// TIA Portal V16 export
// export: Created 2022-11-17T11:55:28.2915288Z, ExportSetting WithDefaults, DisplayName Totally Integrated Automation Portal, DisplayVersion V16 Update 6, DisplayName TIA Portal Version Control Interface, DisplayVersion V16 Update 2, DisplayName TIA Portal Openness, DisplayVersion V16 Update 6, DisplayName SINAMICS Startdrive Advanced, DisplayVersion V16 Update 5, DisplayName SINAMICS Startdrive G130, G150, S120, S150, SINAMICS MV, S210, DisplayVersion V16 Update 5, DisplayName SINAMICS Startdrive G110M, G120, G120C, G120D, G120P, G115D, DisplayVersion V16 Update 5, DisplayName STEP 7 Professional, DisplayVersion V16 Update 6, DisplayName STEP 7 Safety, DisplayVersion V16, DisplayName WinCC Advanced, DisplayVersion V16 Update 6
DATA_BLOCK "DB22_DisplayData"   // DB22
{ S7_Optimized_Access := 'FALSE' }
AUTHOR : Robopac
VERSION : 0.0
// stored: AutoNumber false, IsOnlyStoredInLoadMemory false, IsWriteProtectedInAS false
   VAR RETAIN
      dbx0_0 : Bool := FALSE;   // Technoplat manual(Display): Table rotation forward
      dbx0_1 : Bool := FALSE;   // Technoplat manual(Display): Spool carriage upward
      dbx0_2 : Bool := FALSE;   // Technoplat manual(Display): Spool carriage downward
      dbx0_3 : Bool := FALSE;   // Technoplat manual(Display): Pressure plate upward/downward
      dbx0_4 : Bool := FALSE;   // Technoplat manual(Display): Pallet lifter upward/downward
      dbx0_5 : Bool := FALSE;   // Technoplat manual(Display): Rope unit open/close
      dbx0_6 : Bool := FALSE;   // Technoplat manual(Display): Prestretch
      dbx0_7 : Bool := FALSE;   // Technoplat manual(Display): Spool carriage to film broken position
      dbx1_0 : Bool := FALSE;   // Clamp manual(Display): Clamp upward/downward
      dbx1_1 : Bool := FALSE;   // Clamp manual(Display): Welder unit upward/downward
      dbx1_2 : Bool := FALSE;   // Clamp manual(Display): Welder contrast upward/downward
      dbx1_3 : Bool := FALSE;   // Clamp manual(Display): Clamp carriage forward/backward
      dbx1_4 : Bool := FALSE;   // Clamp manual(Display): Clamp open/close
      dbx1_5 : Bool := FALSE;   // Clamp manual(Display): Cut and welder arm forward/backward
      dbx1_6 : Bool := FALSE;   // Clamp manual(Display): Welder unit forward/backward
      dbx1_7 : Bool := FALSE;   // Clamp manual(Display):
      dbx2_0 : Bool := FALSE;   // Top manual(Display): Top carriage upward
      dbx2_1 : Bool := FALSE;   // Top manual(Display): Top carriage downward
      dbx2_2 : Bool := FALSE;   // Top manual(Display): Top carriage forward
      dbx2_3 : Bool := FALSE;   // Top manual(Display): Top carriage backward
      dbx2_4 : Bool := FALSE;   // Top manual(Display): Opening/closing clamp to pull top film
      dbx2_5 : Bool := FALSE;   // Top manual(Display): Opening/closing clamp to block top film
      dbx2_6 : Bool := FALSE;   // Top manual(Display): Top film cutter forward/backward
      dbx2_7 : Bool := FALSE;   // Top manual(Display): Arm rotation to phase 2 sensor for top
      dbx3_0 : Bool := FALSE;   // Technoplat manual (Display): Rotation to unload
      dbx3_1 : Bool := FALSE;   // Technoplat manual (Display): Rotation to 0
      dbx3_2 : Bool := FALSE;   // Technoplat manual (Display): Rotation to load
      dbx3_3 : Bool := FALSE;
      dbx3_4 : Bool := FALSE;   // Technoplat manual(Display): Rope unit lower open/close
      dbx3_5 : Bool := FALSE;
      dbx3_6 : Bool := FALSE;
      dbx3_7 : Bool := FALSE;
      dbx4_0 : Bool := FALSE;   // Conveyor manual(Display): CMD PRESSED
      dbx4_1 : Bool := FALSE;   // Conveyor manual(Display): Load CM [p18]
      dbx4_2 : Bool := FALSE;   // Conveyor manual(Display): Unload CM [p18]
      dbx4_3 : Bool := FALSE;   // Conveyor manual(Display): RESET ENCODER
      dbx4_4 : Bool := FALSE;   // Conveyor manual(Display): Load CM [Sysdata]
      dbx4_5 : Bool := FALSE;   // Conveyor manual(Display): [not used]
      dbx4_6 : Bool := FALSE;   // Conveyor manual(Display): CM backward slow
      dbx4_7 : Bool := FALSE;   // Conveyor manual(Display): CM forward slow
      dbb5 : Byte := 16#09;   // Conveyor manual operation
      dbx6_0 : Bool := FALSE;   // Manual Signal(Display): Pallet ready in infeed (Input)
      dbx6_1 : Bool := FALSE;   // Manual Signal(Display): Ready to receive pallet infeed (Output)
      dbx6_2 : Bool := FALSE;   // Manual Signal(Display): End of transfer pallet infeed (Output)
      dbx6_3 : Bool := FALSE;   // Manual Signal(Display): Pallet ready in outfeed (Output)
      dbx6_4 : Bool := FALSE;   // Manual Signal(Display): Ready to receive pallet outfeed (Input)
      dbx6_5 : Bool := FALSE;   // Manual Signal(Display): End of transfer pallet outfeed (Input)
      dbx6_6 : Bool := FALSE;   // Manual Signal(Display): Start wrapping signal (Input)
      dbx6_7 : Bool := FALSE;   // Manual Signal(Display): Customer conveyor stopped signal (Input)
      dbx7_0 : Bool := FALSE;   // Manual Signal(Display): Machine in position signal (Output)
      dbx7_1 : Bool := FALSE;   // Manual Signal(Display): Wrapp ended signal (Output)
      dbx7_2 : Bool := FALSE;   // Manual Signal(Display): Pallet in position for label
      dbx7_3 : Bool := TRUE;   // Manual Signal(Display): Label arm in position for pallet transfer
      dbx7_4 : Bool := FALSE;   // Manual Signal(Display): Label cycle ended
      dbx7_5 : Bool := FALSE;   // Manual Signal(Display): Label fault
      dbx7_6 : Bool := FALSE;
      dbx7_7 : Bool := FALSE;
      dbw8 : Int := 0;
      dbw10 : Int := 0;
      dbw12 : Int := 0;
      dbx14_0 : Bool := FALSE;   // Technoplat manual(Program): Table rotation forward
      dbx14_1 : Bool := FALSE;   // Technoplat manual(Program): Spool carriage upward
      dbx14_2 : Bool := FALSE;   // Technoplat manual(Program): Spool carriage downward
      dbx14_3 : Bool := FALSE;   // Technoplat manual(Program): Pressure plate downward
      dbx14_4 : Bool := FALSE;   // Technoplat manual(Program): Pressure plate upward
      dbx14_5 : Bool := FALSE;   // Technoplat manual(Program): Pallet lifter upward
      dbx14_6 : Bool := FALSE;   // Technoplat manual(Program): Pallet lifter downward
      dbx14_7 : Bool := FALSE;   // Technoplat manual(Program): Rope unit closing
      dbx15_0 : Bool := FALSE;   // Technoplat manual(Program): Rope unit opening
      dbx15_1 : Bool := FALSE;   // Technoplat manual(Program): Prestretch
      dbx15_2 : Bool := FALSE;   // Technoplat manual(Program): Spool carriage to film broken position
      dbx15_3 : Bool := FALSE;   // Technoplat manual(Program): Rope unit Lower closing
      dbx15_4 : Bool := FALSE;   // Technoplat manual(Program): Rope unit Lower opening
      dbx15_5 : Bool := FALSE;   // Technoplat manual(Program): CM Backward slow
      dbx15_6 : Bool := FALSE;   // Technoplat manual(Program): CM Forward slow
      dbx15_7 : Bool := FALSE;   // Technoplat manual(Program):
      dbx16_0 : Bool := FALSE;   // Clamp manual(Program): Clamp upward
      dbx16_1 : Bool := FALSE;   // Clamp manual(Program): Clamp downward
      dbx16_2 : Bool := FALSE;   // Clamp manual(Program): Welder unit upward
      dbx16_3 : Bool := FALSE;   // Clamp manual(Program): Welder unit downward
      dbx16_4 : Bool := FALSE;   // Clamp manual(Program): Welder contrast upward
      dbx16_5 : Bool := FALSE;   // Clamp manual(Program): Welder contrast downward
      dbx16_6 : Bool := FALSE;   // Clamp manual(Program): Clamp carriage forward
      dbx16_7 : Bool := FALSE;   // Clamp manual(Program): Clamp carriage backward
      dbx17_0 : Bool := FALSE;   // Clamp manual(Program): Clamp open
      dbx17_1 : Bool := FALSE;   // Clamp manual(Program): Clamp close
      dbx17_2 : Bool := FALSE;   // Clamp manual(Program): Cut and welder arm forward
      dbx17_3 : Bool := FALSE;   // Clamp manual(Program): Cut and welder arm backward
      dbx17_4 : Bool := FALSE;   // Clamp manual(Program): Welder unit forward
      dbx17_5 : Bool := FALSE;   // Clamp manual(Program): Welder unit backward
      dbx17_6 : Bool := FALSE;   // Clamp manual(Program):
      dbx17_7 : Bool := FALSE;   // Clamp manual(Program):
      dbx18_0 : Bool := FALSE;   // Top manual(Program): Top carriage upward
      dbx18_1 : Bool := FALSE;   // Top manual(Program): Top carriage downward
      dbx18_2 : Bool := FALSE;   // Top manual(Program): Top carriage forward
      dbx18_3 : Bool := FALSE;   // Top manual(Program): Top carriage backward
      dbx18_4 : Bool := FALSE;   // Top manual(Program): Opening clamp to pull top film
      dbx18_5 : Bool := FALSE;   // Top manual(Program): Closing clamp to pull top film
      dbx18_6 : Bool := FALSE;   // Top manual(Program): Opening clamp to block top film
      dbx18_7 : Bool := FALSE;   // Top manual(Program): Closing clamp to block top film
      dbx19_0 : Bool := FALSE;   // Top manual(Program): Top film cutter forward/backward
      dbx19_1 : Bool := FALSE;   // Top manual(Program): Arm rotation to phase 2 sensor for top
      dbx19_2 : Bool := FALSE;   // Technoplat manual(Program): Rotation to unload
      dbx19_3 : Bool := FALSE;   // Technoplat manual(Program): Rotation to 0
      dbx19_4 : Bool := FALSE;   // Technoplat manual(Program): Rotation to load
      dbx19_5 : Bool := FALSE;   // Top manual(Program):
      dbx19_6 : Bool := FALSE;   // Top manual(Program):
      dbx19_7 : Bool := FALSE;   // Top manual(Program):
      dbx20_0 : Bool := FALSE;   // Conveyor manual(Program): Load CM
      dbx20_1 : Bool := FALSE;   // Conveyor manual(Program): Unload CM
      dbx20_2 : Bool := FALSE;   // Conveyor manual(Program): CM backward
      dbx20_3 : Bool := FALSE;   // Conveyor manual(Program): Pos.1
      dbx20_4 : Bool := FALSE;   // Conveyor manual(Program): Pos.2
      dbx20_5 : Bool := FALSE;   // Conveyor manual(Program): Pos.3
      dbx20_6 : Bool := FALSE;   // Conveyor manual(Program): Pos.4
      dbx20_7 : Bool := FALSE;   // Conveyor manual(Program): Pos.5
      dbx21_0 : Bool := FALSE;   // Conveyor manual(Program): Pos.6
      dbx21_1 : Bool := FALSE;   // Conveyor manual(Program): Pos.7
      dbx21_2 : Bool := FALSE;   // Conveyor manual(Program): Pos.8
      dbx21_3 : Bool := FALSE;   // Conveyor manual(Program):
      dbx21_4 : Bool := FALSE;   // Conveyor manual(Program):
      dbx21_5 : Bool := FALSE;   // Conveyor manual(Program):
      dbx21_6 : Bool := FALSE;   // Conveyor manual(Program):
      dbx21_7 : Bool := FALSE;   // Conveyor manual(Program):
      dbx22_0 : Bool := FALSE;   // Manual Signal(Program): Pallet ready in infeed (Input)
      dbx22_1 : Bool := FALSE;   // Manual Signal(Program): Ready to receive pallet infeed (Output)
      dbx22_2 : Bool := FALSE;   // Manual Signal(Program): End of transfer pallet infeed (Output)
      dbx22_3 : Bool := FALSE;   // Manual Signal(Program): Pallet ready in outfeed (Output)
      dbx22_4 : Bool := FALSE;   // Manual Signal(Program): Ready to receive pallet outfeed (Input)
      dbx22_5 : Bool := FALSE;   // Manual Signal(Program): End of transfer pallet outfeed (Input)
      dbx22_6 : Bool := FALSE;   // Manual Signal(Program): Start wrapping (Input)
      dbx22_7 : Bool := FALSE;   // Manual Signal(Program): Customer conveyor stopped (Input)
      dbx23_0 : Bool := FALSE;   // Manual Signal(Program): Machine in position (Output)
      dbx23_1 : Bool := FALSE;   // Manual Signal(Program): Wrapp ended (Output)
      dbx23_2 : Bool := FALSE;   // Manual Signal(Program): Pallet ready for label
      dbx23_3 : Bool := TRUE;   // Manual Signal(Program): Label arm in position for pallet transfer
      dbx23_4 : Bool := FALSE;   // Manual Signal(Program): Label cycle ended
      dbx23_5 : Bool := FALSE;   // Manual Signal(Program): Label fault
      dbx23_6 : Bool := FALSE;
      dbx23_7 : Bool := FALSE;
      dbw24 : Int := 0;
      dbw26 : Int := 0;
      dbw28 : Int := 0;
      dbw30 : Int := 0;
      dbx32_0 : Bool := TRUE;   // Manual(Toggle bit): Pressure plate upward/downward (Technplat)
      dbx32_1 : Bool := TRUE;   // Manual(Toggle bit): Pallet lifter upward/downward (Technplat)
      dbx32_2 : Bool := FALSE;   // Manual(Toggle bit): Clamp upward/downward (Clamp)
      dbx32_3 : Bool := FALSE;   // Manual(Toggle bit): Welder unit upward/downward (Clamp)
      dbx32_4 : Bool := TRUE;   // Manual(Toggle bit): Welder contrast upward/downward (Clamp)
      dbx32_5 : Bool := FALSE;   // Manual(Toggle bit): Rope unit open/close (Technplat)
      dbx32_6 : Bool := FALSE;   // Manual(Toggle bit): Clamp open/close (Clamp)
      dbx32_7 : Bool := FALSE;   // Manual(Toggle bit): Cut and welder arm forward/backward (Clamp)
      dbx33_0 : Bool := TRUE;   // Manual(Toggle bit): Opening/closing clamp to pull top film (Top)
      dbx33_1 : Bool := TRUE;   // Manual(Toggle bit): Opening/closing clamp to block top film (Top)
      dbx33_2 : Bool := TRUE;   // Manual(Toggle bit): Welder unit forward/backward (Clamp)
      dbx33_3 : Bool := FALSE;   // Manual(Toggle bit): Clamp carriage forward/backward (Clamp)
      dbx33_4 : Bool := FALSE;   // Manual(Toggle bit): Rope unit lower open/close (Technplat)
      dbx33_5 : Bool := FALSE;   // Manual(Toggle bit):
      dbx33_6 : Bool := FALSE;   // Manual(Toggle bit):
      dbx33_7 : Bool := FALSE;   // Manual(Toggle bit):
      dbw34 : Int := 0;
      dbw36 : Int := 0;
      dbx38_0 : Bool := FALSE;   // Diagnostic signal conveyor: Pallet ready in infeed (input)
      dbx38_1 : Bool := TRUE;   // Diagnostic signal conveyor: Ready to receive pallet infeed (Output)
      dbx38_2 : Bool := FALSE;   // Diagnostic signal conveyor: End of transfer pallet infeed (Output)
      dbx38_3 : Bool := FALSE;   // Diagnostic signal conveyor: Ready to receive pallet in outfeed (Input)
      dbx38_4 : Bool := FALSE;   // Diagnostic signal conveyor: End of transfer pallet outfeed (Input)
      dbx38_5 : Bool := FALSE;   // Diagnostic signal conveyor: Pallet ready in outfeed (Output)
      dbx38_6 : Bool := FALSE;   // Diagnostic signal conveyor: Start wrapping (Input)
      dbx38_7 : Bool := FALSE;   // Diagnostic signal conveyor: Customer conveyor stopped (Input)
      dbx39_0 : Bool := FALSE;   // Diagnostic signal conveyor: Machine in position (Output)
      dbx39_1 : Bool := FALSE;   // Diagnostic signal conveyor: Wrapp ended (Output)
      dbx39_2 : Bool := FALSE;   // Diagnostic signal conveyor: Pallet ready for label
      dbx39_3 : Bool := TRUE;   // Diagnostic signal conveyor: Label arm in position for pallet transit
      dbx39_4 : Bool := FALSE;   // Diagnostic signal conveyor: Label cycle ended
      dbx39_5 : Bool := FALSE;   // Diagnostic signal conveyor: Label fault
      dbw40 : Int := 1;   // Machine status
      dbd42 : DInt := 4;   // Worked hours
      dbd46 : DInt := 95;   // Partial counter for wrapped pallet
      dbd50 : DInt := 163;   // Counter for wrapped pallet
      dbd54 : DInt := 0;
      dbw58 : Int := 21;   // Seconds for worked hours counter
      dbw60 : Int := 36;   // Minutes for worked hours counter
      dbw62 : Int := 0;   // Arm rotation speed (rpm)
      dbw64 : Int := 0;   // Arm rotation speed (rpm)
      dbw66 : Int := 15;   // Number of revolution done on last pallet
      dbw68 : Int := 777;   // Wrapping cycle time
      dbw70 : Int := 22482;   // Wrapping cycle + pallet transfer time
      dbw72 : Int := 10;   // Pallet per hour (Productivity)
      dbw74 : Int := 0;   // Film weight every wrapping cycle (g*10)
      dbw76 : Int := 0;   // Film force for film weight value
      dbw78 : Int := 0;   // Film prestretch for film weight value
      dbw80 : Int := 0;
      dbw82 : Int := 0;
      dbw84 : Int := 0;
      dbw86 : Int := 0;
      dbw88 : Int := 0;
      dbw90 : Int := 0;
      dbw92 : Int := 0;
      dbw94 : Int := 0;
      dbw96 : Int := 0;
      dbw98 : Int := 0;
   END_VAR
BEGIN
END_DATA_BLOCK
